// Mitsubishi GX Works2 project: PLC_GROUP16   PLC: FX3G
// PLC

// global labels: Global1
VAR_GLOBAL CONSTANT
  OrangeConst : REAL := 70.0;
  ClementineConst : REAL := 130.0;
END_VAR
VAR_GLOBAL
  INV_Orange AT D1100 : REAL;
  INV_Clementine AT D1110 : REAL;
  EnterLamp AT Y010 : BOOL;
  Day_Started AT X010 : BOOL;
END_VAR
VAR_GLOBAL CONSTANT
  PomelaConst : REAL := 160.0;
END_VAR
VAR_GLOBAL
  INV_Pomela AT D1115 : REAL;
END_VAR
VAR_GLOBAL CONSTANT
  MinOrangeAmount : REAL;
END_VAR
VAR_GLOBAL
  CheckLamp AT M7 : BOOL;
  Switch1 AT X002 : BOOL;
  WatchTimer AT TC200 : BOOL;
END_VAR
VAR_GLOBAL CONSTANT
  ThreeSec : INT := 300;
END_VAR
VAR_GLOBAL
  TS_200 AT TS200 : BOOL;
  WashLamp AT Y005 : BOOL;
END_VAR
VAR_GLOBAL CONSTANT
  MaxOrangeWash : REAL := 100.0;
END_VAR
VAR_GLOBAL
  OrangeWashingCont AT D1150 : REAL;
END_VAR
VAR_GLOBAL CONSTANT
  DivideBy2 : REAL := 2;
END_VAR
VAR_GLOBAL
  HelpIndicator1 AT M10 : BOOL;
  ClementineWashingCont AT D1155 : REAL;
  PomelaWashingCont AT D1160 : REAL;
  HelpIndicator2 AT M12 : BOOL;
  X1_Switch AT X001 : BOOL;
  X2_Switch AT X002 : BOOL;
  Y1_Lamp AT Y001 : BOOL;
  Indicator_Squeez AT M14 : BOOL;
  SqueezingCont AT D1165 : REAL;
  IsSqueezingContFull AT M16 : BOOL;
  SqueezingFull_Counter AT CC10 : BOOL;
  CS_10 AT CS10 : BOOL;
END_VAR
VAR_GLOBAL CONSTANT
  Const1 : INT := 1;
END_VAR
VAR_GLOBAL
  Indicator3 AT M18 : BOOL;
  M_20 AT M20 : BOOL;
  M_22 AT M22 : BOOL;
END_VAR
VAR_GLOBAL CONSTANT
  Const_0 : REAL;
END_VAR
VAR_GLOBAL
  X_11 AT X011 : BOOL;
  X11DoublePress_Counter AT CC10 : BOOL;
END_VAR
VAR_GLOBAL CONSTANT
  Const2 : INT := 2;
END_VAR
VAR_GLOBAL
  Phase3_Timer AT TC210 : BOOL;
  TS_210 AT TS210 : BOOL;
END_VAR
VAR_GLOBAL CONSTANT
  HalfSec : INT := 50;
END_VAR
VAR_GLOBAL
  HelpBlink1 AT M1 : BOOL;
  Y2_Lamp AT Y002 : BOOL;
  Y3_Lamp AT Y003 : BOOL;
  HalfSec_Timer AT TC202 : BOOL;
  TS_202 AT TS202 : BOOL;
  HalfSec_Timer2 AT TC204 : BOOL;
  TS_204 AT TS204 : BOOL;
  JuiceCont AT D1170 : REAL;
  IsInJuiceCont AT M5 : BOOL;
END_VAR
VAR_GLOBAL CONSTANT
  Const_5 : REAL := 5.0;
  Const_1 : REAL := 1.0;
END_VAR
VAR_GLOBAL
  Analog_Input1 AT D8280 : INT;
  Analog_Input2 AT D8281 : INT;
  Quality_Grade AT D1180 : REAL;
  Is_Quality_Good AT M6 : BOOL;
  X_3 AT X003 : BOOL;
  Quality_Timer AT TC216 : BOOL;
END_VAR
VAR_GLOBAL CONSTANT
  Five_Sec : INT := 500;
END_VAR
VAR_GLOBAL
  TS_212 AT TS212 : BOOL;
  Y4_Lamp AT Y004 : BOOL;
  StorageCont AT D1185 : REAL;
  Bad_Quality_Counter AT CC14 : BOOL;
  CS_14 AT CS14 : BOOL;
END_VAR
VAR_GLOBAL CONSTANT
  Const_1_Analog : REAL := 1.0;
  Const_5_Analog : REAL := 5.0;
END_VAR
VAR_GLOBAL
  Y5_Lamp AT Y005 : BOOL;
  Y0_Lamp AT Y000 : BOOL;
  Real_Analog_Input AT D1190 : REAL;
END_VAR
VAR_GLOBAL CONSTANT
  DivBy400 : REAL := 400;
END_VAR
VAR_GLOBAL
  TS_216 AT TS216 : BOOL;
  Juice_Is_Ready AT M19 : BOOL;
END_VAR
VAR_GLOBAL CONSTANT
  Bottle_Size : REAL := 1.5;
END_VAR
VAR_GLOBAL
  Bottle2 AT X004 : BOOL;
  Bottle1 AT X006 : BOOL;
  X_7 AT X007 : BOOL;
  M_21 AT M21 : BOOL;
  Bottle1_Fill AT M23 : BOOL;
END_VAR
VAR_GLOBAL CONSTANT
  Bottle1_Size : REAL := 1.0;
  Const_10 : REAL := 10.0;
END_VAR
VAR_GLOBAL
  Analog_Output AT D8282 : INT;
END_VAR
VAR_GLOBAL CONSTANT
  Mul_For_Analog : INT := 400;
END_VAR
VAR_GLOBAL
  Bottle2_Fill AT M3 : BOOL;
END_VAR
VAR_GLOBAL CONSTANT
  Bottle_Size2 : REAL := 2.0;
END_VAR
VAR_GLOBAL
  X_0 AT X000 : BOOL;
  Day_End AT M9 : BOOL;
  Day_Is_Going AT M24 : BOOL;
  Condition_Is_OK AT M26 : BOOL;
  Condition_Is_not_OK1 AT M28 : BOOL;
  End_Day_Timer1 AT TC206 : BOOL;
  TS_206 AT TS206 : BOOL;
  Finish_Bottling AT M2 : BOOL;
END_VAR
VAR_GLOBAL CONSTANT
  Const_0Word : INT;
END_VAR
VAR_GLOBAL
  CheckCheck111111 AT M100 : BOOL;
  Orange_Initial_Quantity AT D1280 : REAL;
  Clementine_Init_Quantity AT D1285 : REAL;
  Pomela_Init_Quantity AT D1290 : REAL;
  Is_Squeez_Full AT M22 : BOOL;
END_VAR

// task Task_01 (event TRUE, interval 0, priority 31): POU_01

PROGRAM POU_01
(* structured ladder/FBD written out as ST: instructions are called as NAME(EN, inputs, outputs); _pN, _eN, _tN stand for wires *)
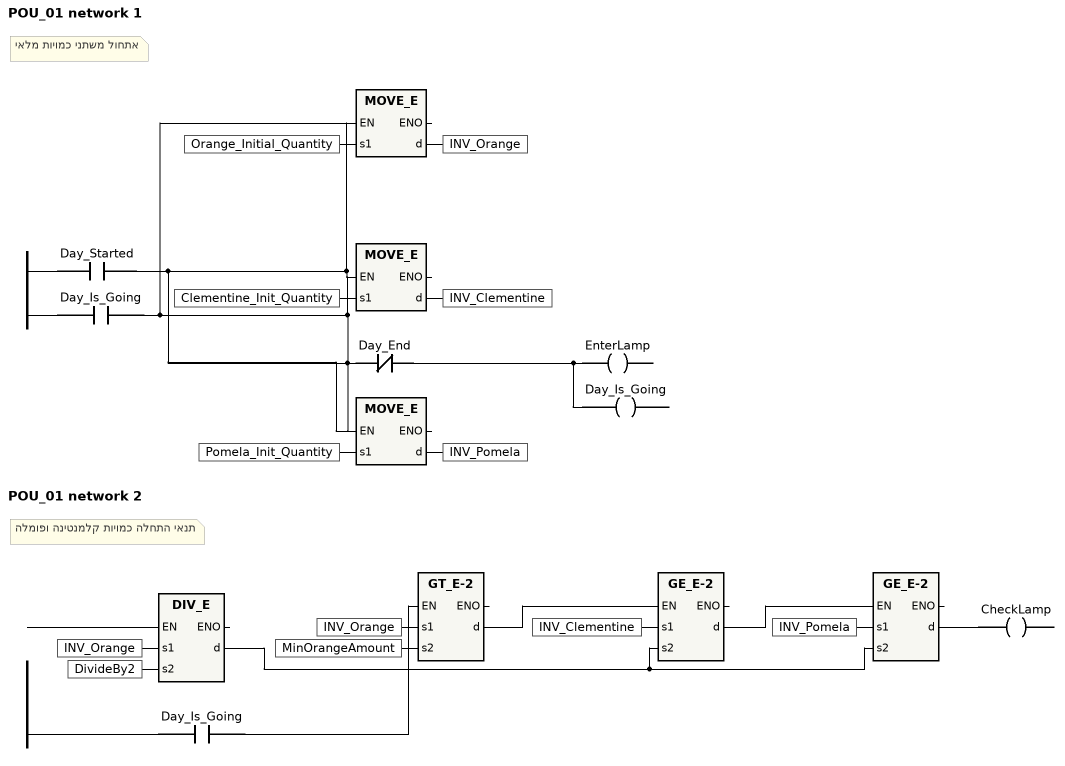
(* network 1 *)
(* אתחול משתני כמויות מלאי *)
_p1 := Day_Started OR Day_Is_Going;
MOVE_E(_p1, Orange_Initial_Quantity, INV_Orange);
MOVE_E(_p1, Clementine_Init_Quantity, INV_Clementine);
MOVE_E(_p1, Pomela_Init_Quantity, INV_Pomela);
_p2 := _p1 AND NOT Day_End;
EnterLamp := _p2;
Day_Is_Going := _p2;
(* network 2 *)
(* תנאי התחלה כמויות קלמנטינה ופומלה *)
GT_E(Day_Is_Going, INV_Orange, MinOrangeAmount, _t1);
DIV_E(TRUE, INV_Orange, DivideBy2, _t2);
GE_E(_t1, INV_Clementine, _t2, _t3);
GE_E(_t3, INV_Pomela, _t2, _t4);
CheckLamp := _t4;
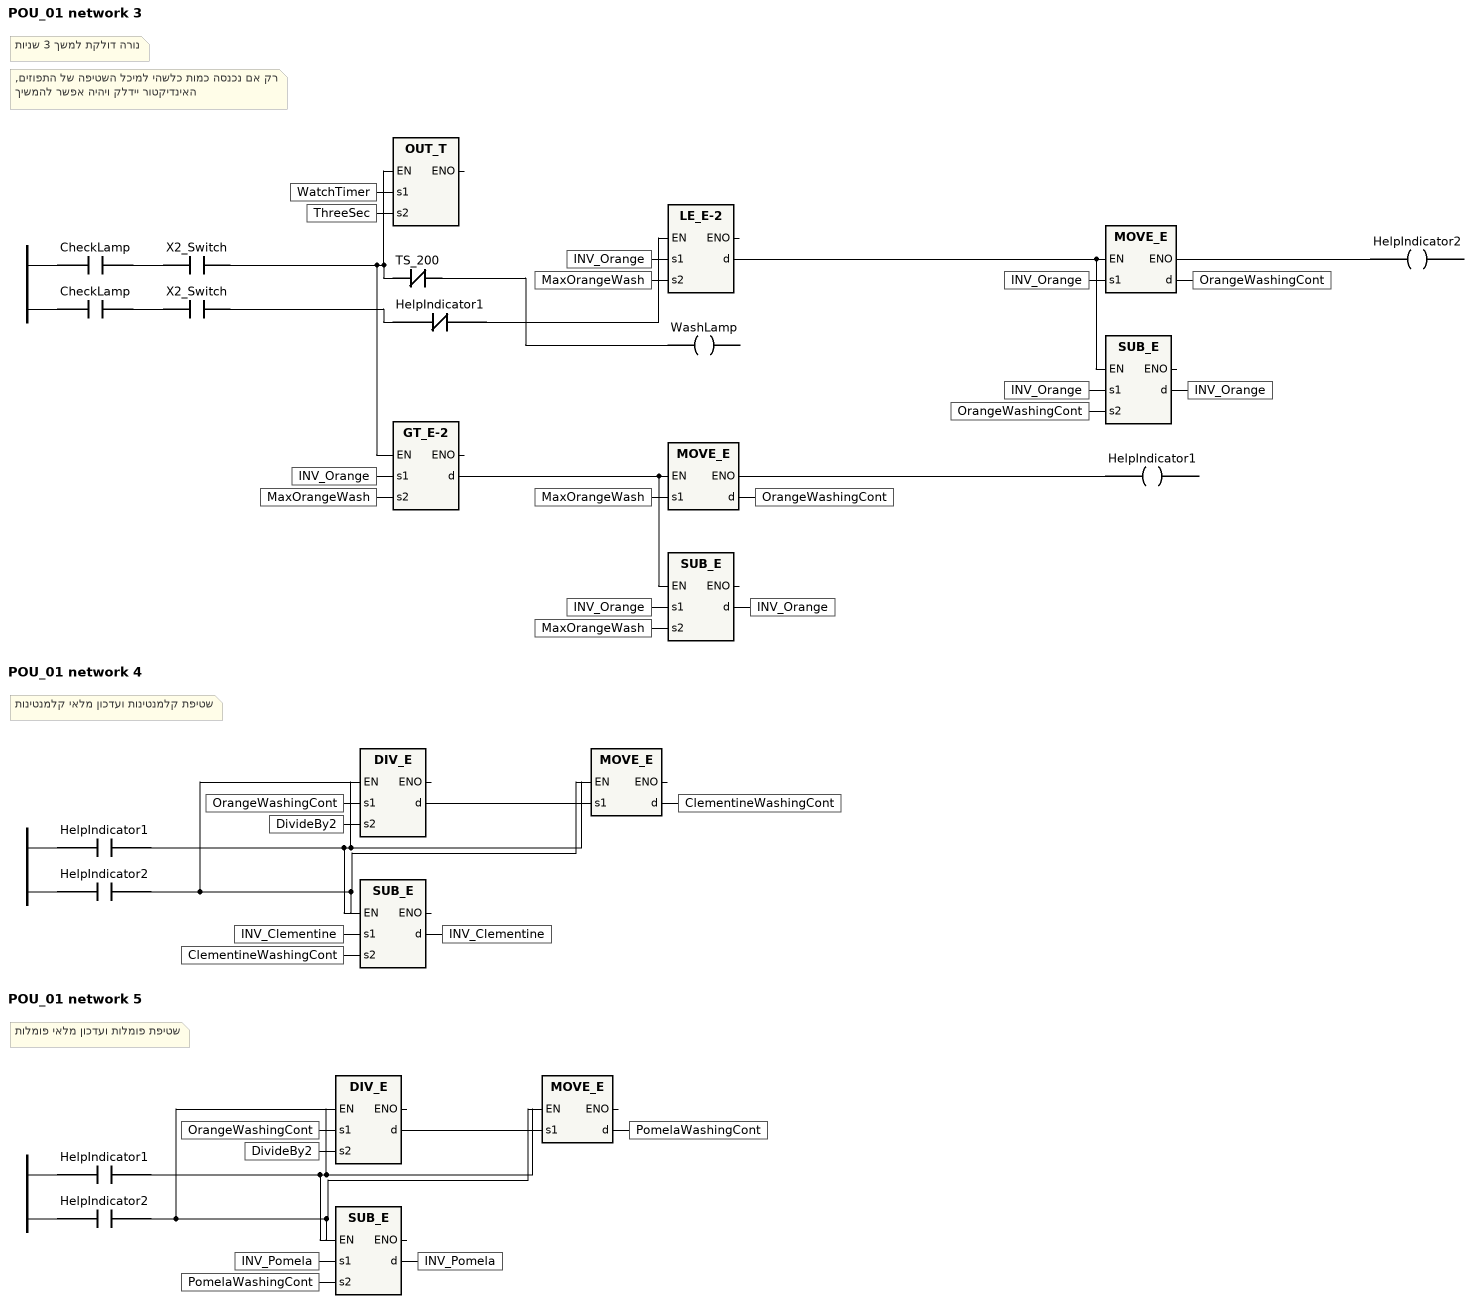
(* network 3 *)
(* נורה דולקת למשך 3 שניות *)
(* רק אם נכנסה כמות כלשהי למיכל השטיפה של התפוזים, האינדיקטור יידלק ויהיה אפשר להמשיך *)
_p1 := CheckLamp AND X2_Switch;
WashLamp := _p1 AND NOT TS_200;
OUT_T(_p1, WatchTimer, ThreeSec);
GT_E(_p1, INV_Orange, MaxOrangeWash, _t2);
_e3 := MOVE_E(_t2, MaxOrangeWash, OrangeWashingCont);
HelpIndicator1 := _e3;
SUB_E(_t2, INV_Orange, MaxOrangeWash, INV_Orange);
LE_E(CheckLamp AND X2_Switch AND NOT HelpIndicator1, INV_Orange, MaxOrangeWash, _t4);
_e5 := MOVE_E(_t4, INV_Orange, OrangeWashingCont);
HelpIndicator2 := _e5;
SUB_E(_t4, INV_Orange, OrangeWashingCont, INV_Orange);
(* network 4 *)
(* שטיפת קלמנטינות ועדכון מלאי קלמנטינות *)
_p1 := HelpIndicator1 OR HelpIndicator2;
DIV_E(_p1, OrangeWashingCont, DivideBy2, _t2);
MOVE_E(_p1, _t2, ClementineWashingCont);
SUB_E(_p1, INV_Clementine, ClementineWashingCont, INV_Clementine);
(* network 5 *)
(* שטיפת פומלות ועדכון מלאי פומלות *)
_p1 := HelpIndicator1 OR HelpIndicator2;
DIV_E(_p1, OrangeWashingCont, DivideBy2, _t2);
MOVE_E(_p1, _t2, PomelaWashingCont);
SUB_E(_p1, INV_Pomela, PomelaWashingCont, INV_Pomela);
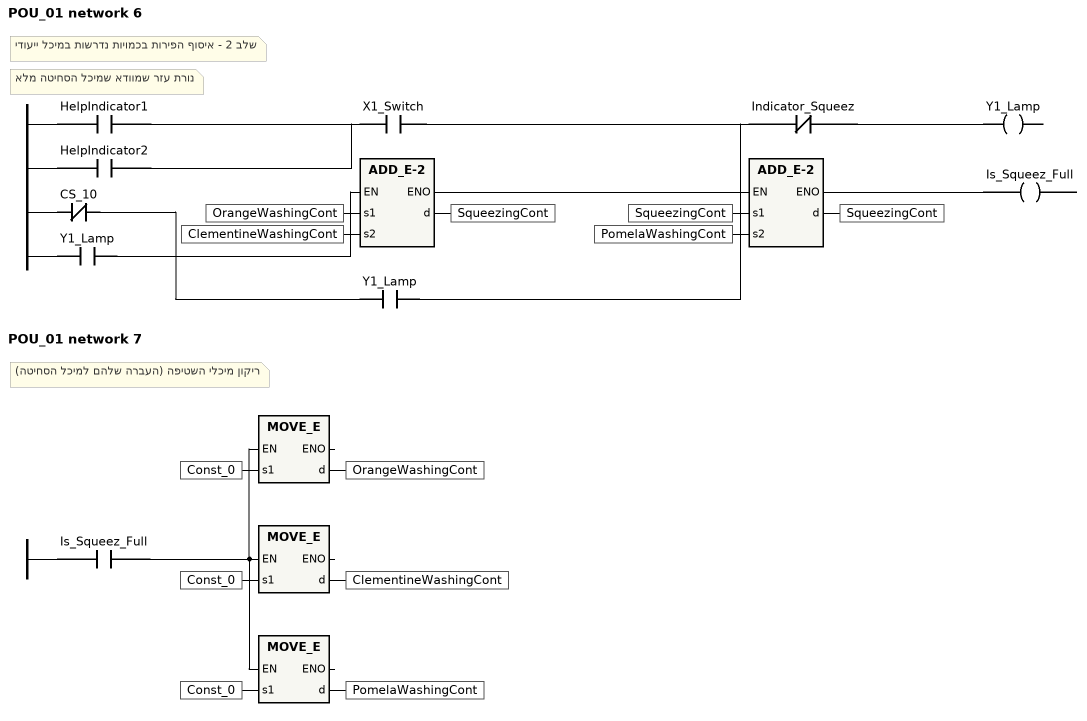
(* network 6 *)
(* שלב 2 - איסוף הפירות בכמויות נדרשות במיכל ייעודי *)
(* נורת עזר שמוודא שמיכל הסחיטה מלא *)
Y1_Lamp := (((HelpIndicator1 OR HelpIndicator2) AND X1_Switch) OR (NOT CS_10 AND Y1_Lamp)) AND NOT Indicator_Squeez;
_e1 := ADD_E(Y1_Lamp, OrangeWashingCont, ClementineWashingCont, SqueezingCont);
_e2 := ADD_E(_e1, SqueezingCont, PomelaWashingCont, SqueezingCont);
Is_Squeez_Full := _e2;
(* network 7 *)
(* ריקון מיכלי השטיפה (העברה שלהם למיכל הסחיטה) *)
MOVE_E(Is_Squeez_Full, Const_0, OrangeWashingCont);
MOVE_E(Is_Squeez_Full, Const_0, ClementineWashingCont);
MOVE_E(Is_Squeez_Full, Const_0, PomelaWashingCont);
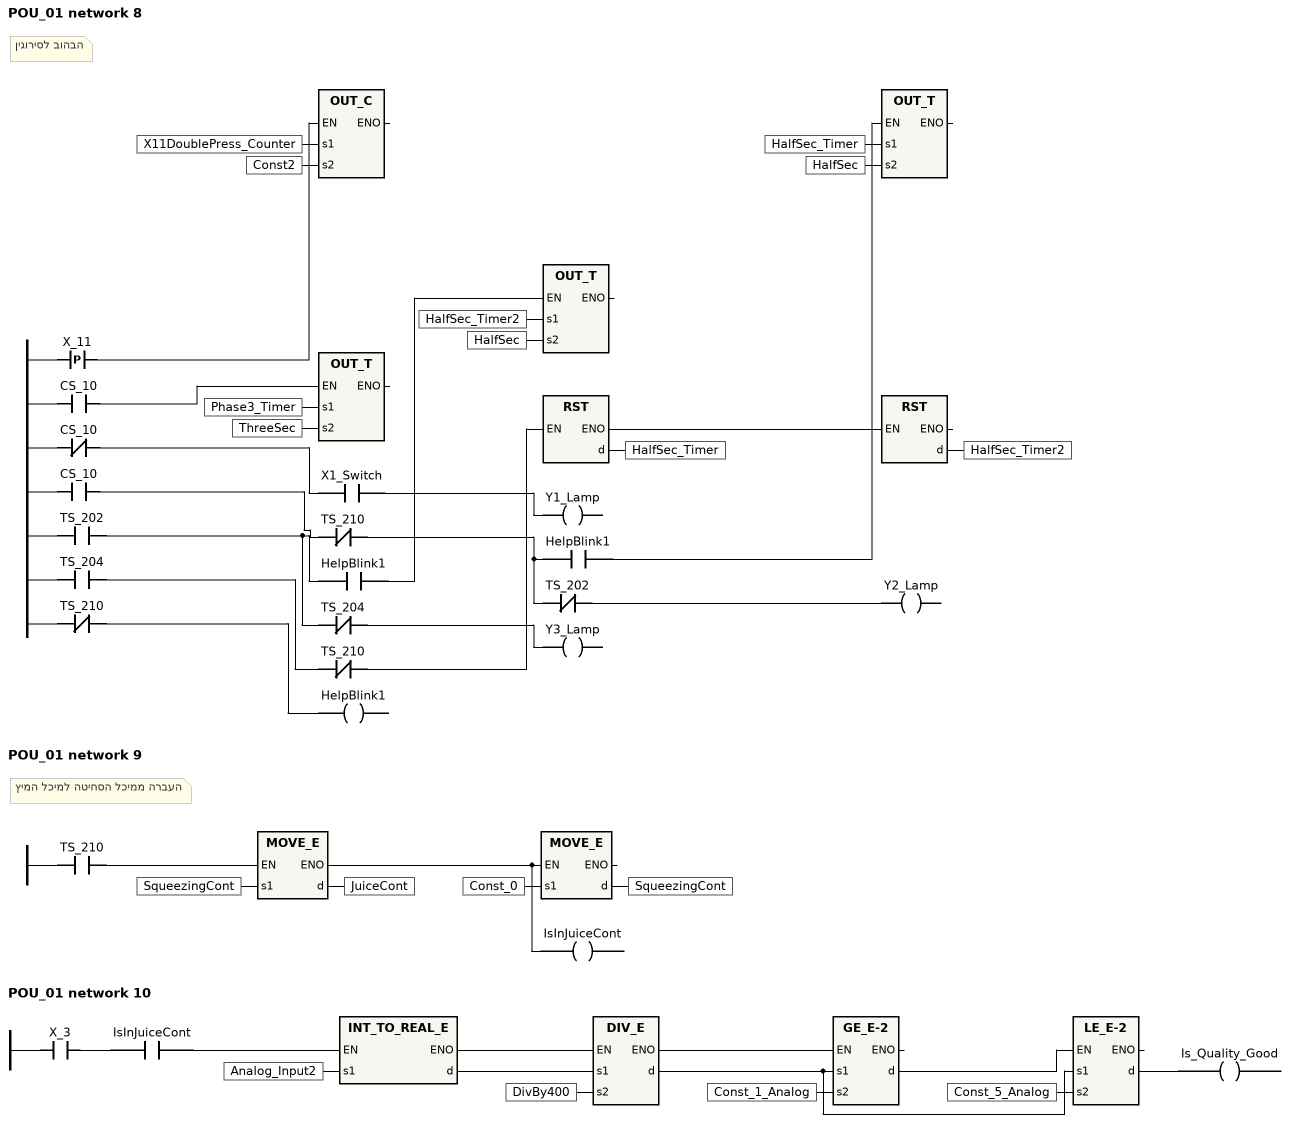
(* network 8 *)
(* הבהוב לסירוגין *)
OUT_C(LDP(TRUE, X_11), X11DoublePress_Counter, Const2);
OUT_T(CS_10, Phase3_Timer, ThreeSec);
Y1_Lamp := NOT CS_10 AND X1_Switch;
_p1 := CS_10 AND NOT TS_210;
OUT_T(_p1 AND HelpBlink1, HalfSec_Timer, HalfSec);
Y2_Lamp := _p1 AND NOT TS_202;
OUT_T(TS_202 AND HelpBlink1, HalfSec_Timer2, HalfSec);
Y3_Lamp := TS_202 AND NOT TS_204;
_e2 := RST(TS_204 AND NOT TS_210, HalfSec_Timer);
RST(_e2, HalfSec_Timer2);
HelpBlink1 := NOT TS_210;
(* network 9 *)
(* העברה ממיכל הסחיטה למיכל המיץ *)
_e1 := MOVE_E(TS_210, SqueezingCont, JuiceCont);
IsInJuiceCont := _e1;
MOVE_E(_e1, Const_0, SqueezingCont);
(* network 10 *)
_e2 := INT_TO_REAL_E(X_3 AND IsInJuiceCont, Analog_Input2, _t1);
_e4 := DIV_E(_e2, _t1, DivBy400, _t3);
GE_E(_e4, _t3, Const_1_Analog, _t5);
LE_E(_t5, _t3, Const_5_Analog, _t6);
Is_Quality_Good := _t6;
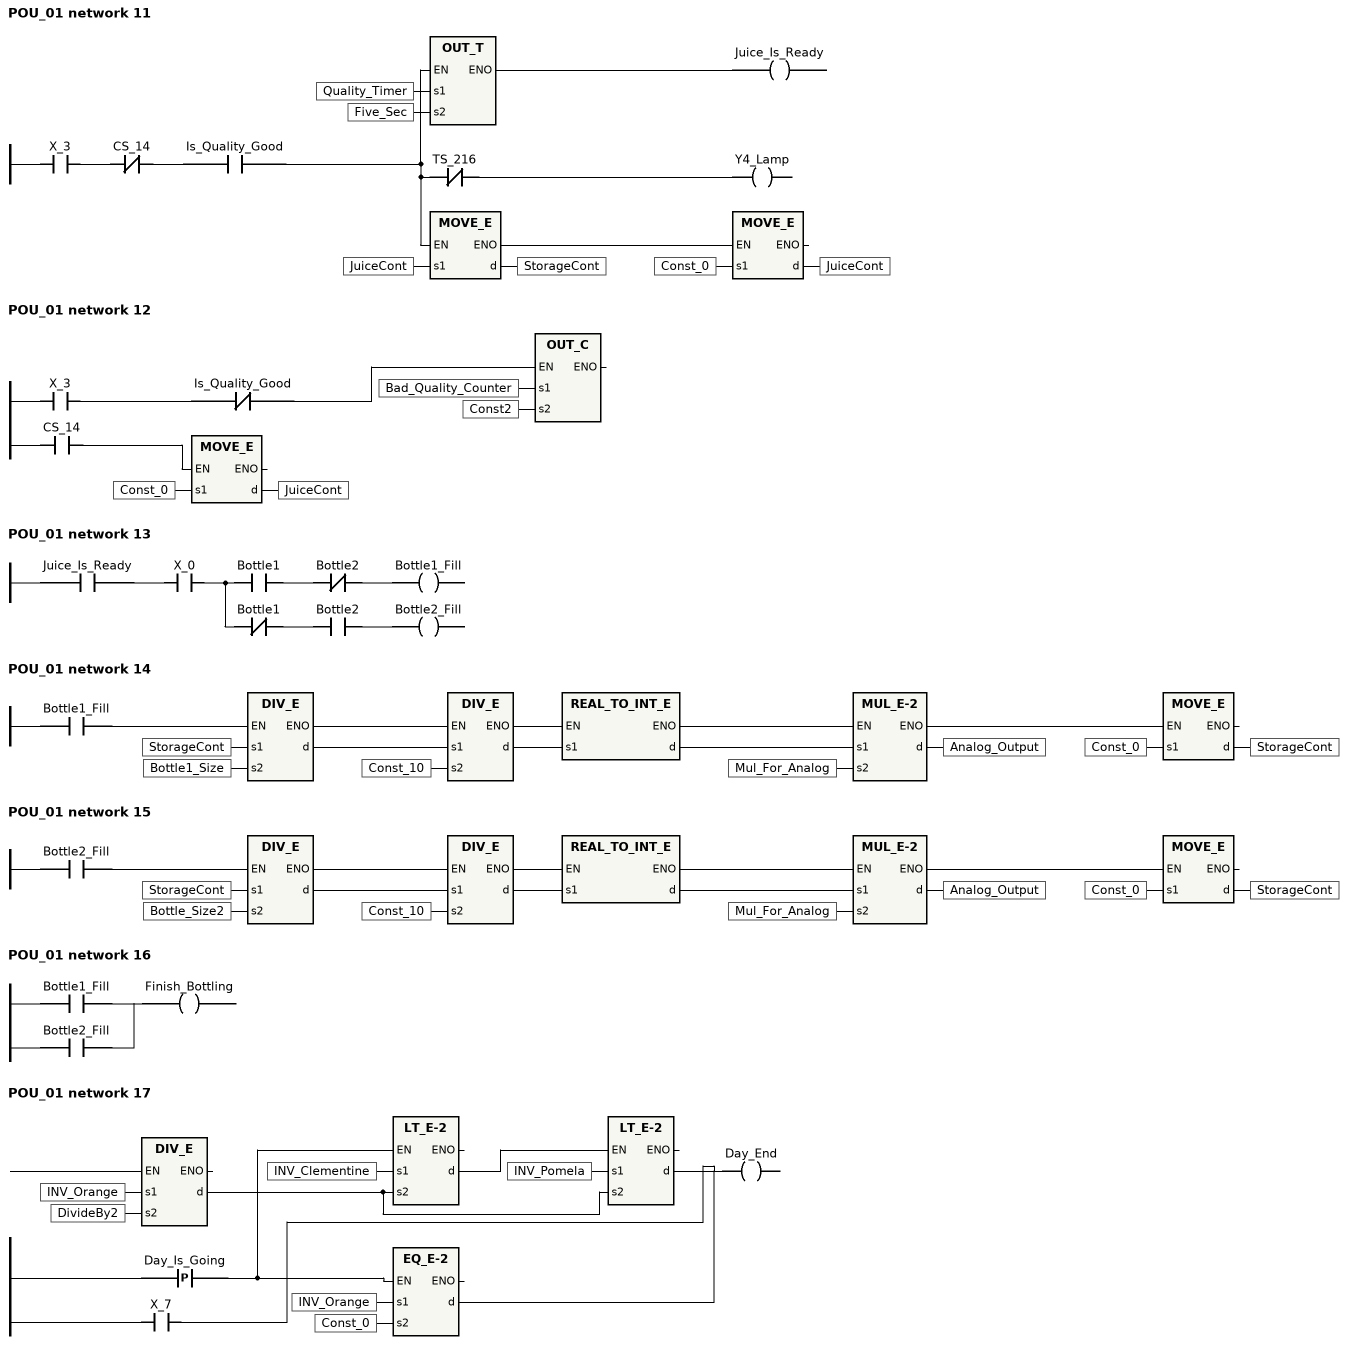
(* network 11 *)
_p1 := X_3 AND NOT CS_14 AND Is_Quality_Good;
_e2 := OUT_T(_p1, Quality_Timer, Five_Sec);
Juice_Is_Ready := _e2;
Y4_Lamp := _p1 AND NOT TS_216;
_e3 := MOVE_E(_p1, JuiceCont, StorageCont);
MOVE_E(_e3, Const_0, JuiceCont);
(* network 12 *)
OUT_C(X_3 AND NOT Is_Quality_Good, Bad_Quality_Counter, Const2);
MOVE_E(CS_14, Const_0, JuiceCont);
(* network 13 *)
_p1 := Juice_Is_Ready AND X_0;
Bottle1_Fill := _p1 AND Bottle1 AND NOT Bottle2;
Bottle2_Fill := _p1 AND NOT Bottle1 AND Bottle2;
(* network 14 *)
_e2 := DIV_E(Bottle1_Fill, StorageCont, Bottle1_Size, _t1);
_e4 := DIV_E(_e2, _t1, Const_10, _t3);
_e6 := REAL_TO_INT_E(_e4, _t3, _t5);
_e7 := MUL_E(_e6, _t5, Mul_For_Analog, Analog_Output);
MOVE_E(_e7, Const_0, StorageCont);
(* network 15 *)
_e2 := DIV_E(Bottle2_Fill, StorageCont, Bottle_Size2, _t1);
_e4 := DIV_E(_e2, _t1, Const_10, _t3);
_e6 := REAL_TO_INT_E(_e4, _t3, _t5);
_e7 := MUL_E(_e6, _t5, Mul_For_Analog, Analog_Output);
MOVE_E(_e7, Const_0, StorageCont);
(* network 16 *)
Finish_Bottling := Bottle1_Fill OR Bottle2_Fill;
(* network 17 *)
_p1 := LDP(TRUE, Day_Is_Going);
EQ_E(_p1, INV_Orange, Const_0, _t2);
DIV_E(TRUE, INV_Orange, DivideBy2, _t3);
LT_E(_p1, INV_Clementine, _t3, _t4);
LT_E(_t4, INV_Pomela, _t3, _t5);
Day_End := _t2 OR _t5 OR X_7;
END_PROGRAM
